PROGRAM PRG_Roughing
VAR
END_VAR

// Roughing devices

qRIXS_ROUGH_GPI_02();			// Roughing guage near BL 


//VRC 02	
qRIXS_ROUGH_VRC_02(i_xExtILK_OK := TRUE, i_xOverrideMode := xSystemOverrideMode, iq_stValve => );

//VRC 01
qRIXS_ROUGH_VRC_01(i_xExtILK_OK := TRUE, i_xOverrideMode := xSystemOverrideMode, iq_stValve => );

END_PROGRAM

(* stored: Version 1.1.0.1, ProductVersion 3.1.4022.18
   POU PRG_Roughing: Id {9373ef9e-5e95-4b75-81c2-b0e4a1795889}, SpecialFunc None *)
